Permission is hereby granted, free of charge, to any person obtaining a copy 
of this software and associated documentation files (the "Software"), to deal 
in the Software without restriction, including without limitation the rights 
to use, copy, modify, merge, publish, distribute, sublicense, and/or sell 
copies of the Software, and to permit persons to whom the Software is 
furnished to do so, subject to the following conditions:

The above copyright notice and this permission notice shall be included in 
all copies or substantial portions of the Software.

THE SOFTWARE IS PROVIDED "AS IS", WITHOUT WARRANTY OF ANY KIND, EXPRESS OR 
IMPLIED, INCLUDING BUT NOT LIMITED TO THE WARRANTIES OF MERCHANTABILITY, 
FITNESS FOR A PARTICULAR PURPOSE AND NONINFRINGEMENT. IN NO EVENT SHALL THE 
AUTHORS OR COPYRIGHT HOLDERS BE LIABLE FOR ANY CLAIM, DAMAGES OR OTHER 
LIABILITY, WHETHER IN AN ACTION OF CONTRACT, TORT OR OTHERWISE, ARISING FROM, 
OUT OF OR IN CONNECTION WITH THE SOFTWARE OR THE USE OR OTHER DEALINGS 
IN THE SOFTWARE.
*)
fin := FALSE;
                    
END_ACTION

ACTION TO_DEFAULT_POS_2_active:
                      (*
Copyright (c) 2019 Manuel Goester, Michael Witt, Klaus Kammerer
Institute of Databases and Information Systems, Ulm University, Germany

Permission is hereby granted, free of charge, to any person obtaining a copy 
of this software and associated documentation files (the "Software"), to deal 
in the Software without restriction, including without limitation the rights 
to use, copy, modify, merge, publish, distribute, sublicense, and/or sell 
copies of the Software, and to permit persons to whom the Software is 
furnished to do so, subject to the following conditions:

The above copyright notice and this permission notice shall be included in 
all copies or substantial portions of the Software.

THE SOFTWARE IS PROVIDED "AS IS", WITHOUT WARRANTY OF ANY KIND, EXPRESS OR 
IMPLIED, INCLUDING BUT NOT LIMITED TO THE WARRANTIES OF MERCHANTABILITY, 
FITNESS FOR A PARTICULAR PURPOSE AND NONINFRINGEMENT. IN NO EVENT SHALL THE 
AUTHORS OR COPYRIGHT HOLDERS BE LIABLE FOR ANY CLAIM, DAMAGES OR OTHER 
LIABILITY, WHETHER IN AN ACTION OF CONTRACT, TORT OR OTHERWISE, ARISING FROM, 
OUT OF OR IN CONNECTION WITH THE SOFTWARE OR THE USE OR OTHER DEALINGS 
IN THE SOFTWARE.
*)
// get HR to its default position
// needed, if a job multi / single mode batch job will be executed after ths batch
IF HR.sCBack = FALSE THEN
	HR.mCBackward := TRUE;
ELSE 
	HR.mCBackward := FALSE;
	// set tower vertical position to max UP as well as horizontal position max RIGHT
	IF HR.sHorizontal = FALSE THEN
		HR.mHorizontalRight := TRUE;
	ELSE
		HR.mHorizontalRight := FALSE;
		HR.cX := 0;
	END_IF
	
	IF HR.sVertical = FALSE THEN
		HR.mVerticalUp := TRUE;
	ELSE
		HR.mVerticalUp := FALSE;
		HR.cY := 0;
	END_IF
END_IF

IF HR.sHorizontal AND HR.sVertical AND HR.sCBack THEN
	// finished
	fin := TRUE;
END_IF
                    
END_ACTION
END_PROGRAM

(* Picks up a workpiece Copyright (c) 2019 Manuel Goester, Michael Witt, Klaus Kammerer Institute of Databases and Information Systems, Ulm University, Germany Permission is hereby granted, free of charge, to any person obtaining a copy of this software and associated documentation files (the "Software"), to deal in the Software without restriction, including without limitation the rights to use, copy, modify, merge, publish, distribute, sublicense, and/or sell copies of the Software, and to permit persons to whom the Software is furnished to do so, subject to the following conditions: The above copyright notice and this permission notice shall be included in all copies or substantial portions of the Software. THE SOFTWARE IS PROVIDED "AS IS", WITHOUT WARRANTY OF ANY KIND, EXPRESS OR IMPLIED, INCLUDING BUT NOT LIMITED TO THE WARRANTIES OF MERCHANTABILITY, FITNESS FOR A PARTICULAR PURPOSE AND NONINFRINGEMENT. IN NO EVENT SHALL THE AUTHORS OR COPYRIGHT HOLDERS BE LIABLE FOR ANY CLAIM, DAMAGES OR OTHER LIABILITY, WHETHER IN AN ACTION OF CONTRACT, TORT OR OTHERWISE, ARISING FROM, OUT OF OR IN CONNECTION WITH THE SOFTWARE OR THE USE OR OTHER DEALINGS IN THE SOFTWARE. *)
FUNCTION_BLOCK HR_TAKE_W
  VAR_INPUT
    w : Workpiece;  (* The workpiece *)
  END_VAR
  VAR
    step : INT := 1;
    hr_move : HR_MOVE;
    fin : BOOL := FALSE;
    stepFin : BOOL := FALSE;
  END_VAR

                  fin := FALSE;
CASE step OF
	1:	// forward
		IF NOT(HR.sCFront) THEN
			HR.mCForward := TRUE;
		ELSE
			HR.mCForward := FALSE;
			step := step + 1;
		END_IF
	2:	// up
		hr_move(x := 0, y := -16);
		stepFin := hr_move.fin;
		IF stepFin THEN
			step := step + 1;
			stepFin := FALSE;
		END_IF
	3:	// step 3: back
		IF NOT(HR.sCBack) THEN
			HR.mCBackward := TRUE;
		ELSE
			HR.mCBackward := FALSE;
			step := step + 1;
		END_IF
	4:	// finished
		fin := TRUE;
		step := 1;
		stepFin := FALSE;	
END_CASE
                
END_FUNCTION_BLOCK

(* Moves VG to certain position Copyright (c) 2019 Manuel Goester, Michael Witt, Klaus Kammerer Institute of Databases and Information Systems, Ulm University, Germany Permission is hereby granted, free of charge, to any person obtaining a copy of this software and associated documentation files (the "Software"), to deal in the Software without restriction, including without limitation the rights to use, copy, modify, merge, publish, distribute, sublicense, and/or sell copies of the Software, and to permit persons to whom the Software is furnished to do so, subject to the following conditions: The above copyright notice and this permission notice shall be included in all copies or substantial portions of the Software. THE SOFTWARE IS PROVIDED "AS IS", WITHOUT WARRANTY OF ANY KIND, EXPRESS OR IMPLIED, INCLUDING BUT NOT LIMITED TO THE WARRANTIES OF MERCHANTABILITY, FITNESS FOR A PARTICULAR PURPOSE AND NONINFRINGEMENT. IN NO EVENT SHALL THE AUTHORS OR COPYRIGHT HOLDERS BE LIABLE FOR ANY CLAIM, DAMAGES OR OTHER LIABILITY, WHETHER IN AN ACTION OF CONTRACT, TORT OR OTHERWISE, ARISING FROM, OUT OF OR IN CONNECTION WITH THE SOFTWARE OR THE USE OR OTHER DEALINGS IN THE SOFTWARE. *)
FUNCTION_BLOCK VG_MOVE_TO_POS
  VAR_INPUT
    x : INT;
    y : INT;
    z : INT;
  END_VAR
  VAR
    xFin : BOOL := FALSE;  (* finish flags *)
    yFin : BOOL := FALSE;
    zFin : BOOL := FALSE;
    fin : BOOL := FALSE;
    xAlreadyCounted : BOOL := FALSE;  (* true, if an impulse coming from the motor has been already counted *)
    yAlreadyCounted : BOOL := FALSE;
    zAlreadyCounted : BOOL := FALSE;
  END_VAR

                  fin := FALSE;
// to handle negative counter values
IF VG.cX < 0 THEN
	VG.cX := 0;
END_IF
IF VG.cY < 0 THEN
	VG.cY := 0;
END_IF
IF VG.cZ < 0 THEN
	VG.cZ := 0;
END_IF

// X AXIS (Forward/Backward)
IF VG.cX = x THEN
	// if counter reached demanded position, we're done
	VG.mHorizontalForward := FALSE;
	VG.mHorizontalBackward := FALSE;
	xFin := TRUE;
ELSE
	xFin := FALSE;
	IF VG.cX < x AND NOT(xFin) THEN
		VG.mHorizontalForward := TRUE;
		VG.mHorizontalBackward := FALSE;
		IF VG.encHorizontal AND NOT(xAlreadyCounted) THEN
			VG.cX := VG.cX + 1;
			xAlreadyCounted := TRUE;
		ELSIF NOT(VG.encHorizontal) THEN
			xAlreadyCounted := FALSE;
		END_IF
	ELSIF VG.cX > x AND NOT(xFin) THEN
		VG.mHorizontalForward := FALSE;
		VG.mHorizontalBackward := TRUE;
		IF VG.encHorizontal AND NOT(xAlreadyCounted) THEN
			VG.cX := VG.cX - 1;
			xAlreadyCounted := TRUE;
		ELSIF NOT(VG.encHorizontal) THEN
			xAlreadyCounted := FALSE;
		END_IF
	END_IF
END_IF

// Y AXIS (Up/Down)
IF VG.cY = y THEN
	// if counter reached demanded position, we're done
	VG.mVerticalUp := FALSE;
	VG.mVerticalDown := FALSE;
	yFin := TRUE;
ELSE
	yFin := FALSE;
	IF VG.cY < y AND NOT(yFin) THEN
		VG.mVerticalDown := TRUE;
		VG.mVerticalUp := FALSE;
		IF VG.encVertical AND NOT(yAlreadyCounted) THEN
			VG.cY := VG.cY + 1;
			yAlreadyCounted := TRUE;
		ELSIF NOT(VG.encVertical) THEN
			yAlreadyCounted := FALSE;
		END_IF
	ELSIF VG.cY > y AND NOT(yFin) THEN
		VG.mVerticalUp := TRUE;
		VG.mVerticalDown := FALSE;
		IF VG.encVertical AND NOT(yAlreadyCounted) THEN
			VG.cY := VG.cY - 1;
			yAlreadyCounted := TRUE;
		ELSIF NOT(VG.encVertical) THEN
			yAlreadyCounted := FALSE;
		END_IF
	END_IF
END_IF

// Z AXIS (Rotation)
IF VG.cZ = z THEN
	// if counter reached demanded position, we're done
	VG.mRotationCClockwise := FALSE;
	VG.mRotationClockwise := FALSE;
	zFin := TRUE;
ELSE
	zFin := FALSE;
	IF VG.cZ < z AND NOT(zFin) THEN
		VG.mRotationCClockwise := TRUE;
		VG.mRotationClockwise := FALSE;
		IF VG.encRotation AND NOT(zAlreadyCounted) THEN
			VG.cZ := VG.cZ + 1;
			zAlreadyCounted := TRUE;
		ELSIF NOT(VG.encRotation) THEN
			zAlreadyCounted := FALSE;
		END_IF
	ELSIF VG.cZ > z AND NOT(zFin) THEN
		VG.mRotationCClockwise := FALSE;
		VG.mRotationClockwise := TRUE;
		IF VG.encRotation AND NOT(zAlreadyCounted) THEN
			VG.cZ := VG.cZ - 1;
			zAlreadyCounted := TRUE;
		ELSIF NOT(VG.encRotation) THEN
			zAlreadyCounted := FALSE;
		END_IF
	END_IF
END_IF

// if x and y axis are finsihed, we're done
IF xFin AND yFin AND zFin THEN
	fin := TRUE;
	RETURN;
END_IF
                
END_FUNCTION_BLOCK

(* HR puts down a workpiece at conveyor Copyright (c) 2019 Manuel Goester, Michael Witt, Klaus Kammerer Institute of Databases and Information Systems, Ulm University, Germany Permission is hereby granted, free of charge, to any person obtaining a copy of this software and associated documentation files (the "Software"), to deal in the Software without restriction, including without limitation the rights to use, copy, modify, merge, publish, distribute, sublicense, and/or sell copies of the Software, and to permit persons to whom the Software is furnished to do so, subject to the following conditions: The above copyright notice and this permission notice shall be included in all copies or substantial portions of the Software. THE SOFTWARE IS PROVIDED "AS IS", WITHOUT WARRANTY OF ANY KIND, EXPRESS OR IMPLIED, INCLUDING BUT NOT LIMITED TO THE WARRANTIES OF MERCHANTABILITY, FITNESS FOR A PARTICULAR PURPOSE AND NONINFRINGEMENT. IN NO EVENT SHALL THE AUTHORS OR COPYRIGHT HOLDERS BE LIABLE FOR ANY CLAIM, DAMAGES OR OTHER LIABILITY, WHETHER IN AN ACTION OF CONTRACT, TORT OR OTHERWISE, ARISING FROM, OUT OF OR IN CONNECTION WITH THE SOFTWARE OR THE USE OR OTHER DEALINGS IN THE SOFTWARE. *)
FUNCTION_BLOCK HR_PUT_W_ON_CONVEYOR
  VAR_INPUT
    w : Workpiece;  (* The workpiece *)
  END_VAR
  VAR
    step : INT := 1;
    hr_move : HR_MOVE;
    fin : BOOL := FALSE;
    stepFin : BOOL := FALSE;
  END_VAR

                  CASE step OF
	1:	// forward
		fin := FALSE;	
		IF NOT(HR.sCFront) THEN
			HR.mCForward := TRUE;
		ELSE
			HR.mCForward := FALSE;
			step := step + 1;
		END_IF
	2:	// down
		hr_move(x := 0 , y := 26);
		stepFin := hr_move.fin; 
		IF stepFin THEN
			step := step + 1;
			stepFin := FALSE;
		END_IF
	3:	// finished
		fin := TRUE;
		step := 1;
END_CASE
	
                
END_FUNCTION_BLOCK

(* Picks up a workpiece from conveyor Copyright (c) 2019 Manuel Goester, Michael Witt, Klaus Kammerer Institute of Databases and Information Systems, Ulm University, Germany Permission is hereby granted, free of charge, to any person obtaining a copy of this software and associated documentation files (the "Software"), to deal in the Software without restriction, including without limitation the rights to use, copy, modify, merge, publish, distribute, sublicense, and/or sell copies of the Software, and to permit persons to whom the Software is furnished to do so, subject to the following conditions: The above copyright notice and this permission notice shall be included in all copies or substantial portions of the Software. THE SOFTWARE IS PROVIDED "AS IS", WITHOUT WARRANTY OF ANY KIND, EXPRESS OR IMPLIED, INCLUDING BUT NOT LIMITED TO THE WARRANTIES OF MERCHANTABILITY, FITNESS FOR A PARTICULAR PURPOSE AND NONINFRINGEMENT. IN NO EVENT SHALL THE AUTHORS OR COPYRIGHT HOLDERS BE LIABLE FOR ANY CLAIM, DAMAGES OR OTHER LIABILITY, WHETHER IN AN ACTION OF CONTRACT, TORT OR OTHERWISE, ARISING FROM, OUT OF OR IN CONNECTION WITH THE SOFTWARE OR THE USE OR OTHER DEALINGS IN THE SOFTWARE. *)
FUNCTION_BLOCK HR_TAKE_W_FROM_CONVEYOR
  VAR_INPUT
    w : Workpiece;
  END_VAR
  VAR
    step : INT := 1;
    hr_move : HR_MOVE;
    fin : BOOL := FALSE;
    stepFin : BOOL := FALSE;
  END_VAR

                  fin := FALSE;
CASE step OF
	1:	// forward if not already there
		IF NOT(HR.sCFront) THEN
			HR.mCForward := TRUE;
		ELSE
			HR.mCForward := FALSE;
			step := step + 1;
		END_IF
	2:	// backwards
		IF HR.lbIn THEN
			HR.mCbBackward := TRUE;
		ELSE
			HR.mCbBackward := FALSE;
			step := step + 1; 
		END_IF
	3:	// up
		hr_move(x := 0, y := -26);
		stepFin := hr_move.fin;
		IF stepFin THEN
			step := step + 1;
			stepFin := FALSE;
		END_IF
	4:	// back
		IF NOT(HR.sCBack) THEN
			HR.mCBackward := TRUE;
		ELSE
			HR.mCBackward := FALSE;
			step := step + 1;
		END_IF
	5:	// finished
		fin := TRUE;
		step := 1;
		stepFin := FALSE;
END_CASE
                
END_FUNCTION_BLOCK

(* Function Block for buring a workpiece in furnace w : Workpiece to be burned Copyright (c) 2019 Manuel Goester, Michael Witt, Klaus Kammerer Institute of Databases and Information Systems, Ulm University, Germany Permission is hereby granted, free of charge, to any person obtaining a copy of this software and associated documentation files (the "Software"), to deal in the Software without restriction, including without limitation the rights to use, copy, modify, merge, publish, distribute, sublicense, and/or sell copies of the Software, and to permit persons to whom the Software is furnished to do so, subject to the following conditions: The above copyright notice and this permission notice shall be included in all copies or substantial portions of the Software. THE SOFTWARE IS PROVIDED "AS IS", WITHOUT WARRANTY OF ANY KIND, EXPRESS OR IMPLIED, INCLUDING BUT NOT LIMITED TO THE WARRANTIES OF MERCHANTABILITY, FITNESS FOR A PARTICULAR PURPOSE AND NONINFRINGEMENT. IN NO EVENT SHALL THE AUTHORS OR COPYRIGHT HOLDERS BE LIABLE FOR ANY CLAIM, DAMAGES OR OTHER LIABILITY, WHETHER IN AN ACTION OF CONTRACT, TORT OR OTHERWISE, ARISING FROM, OUT OF OR IN CONNECTION WITH THE SOFTWARE OR THE USE OR OTHER DEALINGS IN THE SOFTWARE. *)
FUNCTION_BLOCK FUR_BURN
  VAR_INPUT
    w : Workpiece;
  END_VAR
  VAR
    step : INT := 1;
    fin : BOOL := FALSE;
    stepFin : BOOL := FALSE;
    timer : TON;
  END_VAR

                  CASE step OF
	1:	// open door and drive workpiece into furnace
		// reset flag
		fin := FALSE;
		FUR.compressor := TRUE;
		FUR.valveFurnanceDoor := TRUE;
		IF FUR.sFurnanceSliderInside = FALSE THEN
			FUR.mFurnanceSliderIn := TRUE;
		ELSE
			FUR.mFurnanceSliderIn := FALSE;
			FUR.state := FUR_State.FUR_WAGON_INSIDE;
			step := step + 1;
		END_IF
	2:	// burn
		IF FUR.state = FUR_State.FUR_WAGON_INSIDE THEN
			//SM.currW.state := StateEnum.AT_FUR_IN_FUR;
			timer(IN:= TRUE, PT := FUR.currWBurner.format.furDuration);
			FUR.valveFurnanceDoor := FALSE;
			IF NOT(timer.Q = FALSE AND timer.IN) THEN
				// reset timer
				timer(IN:= FALSE);
				FUR.compressor := TRUE;
				FUR.valveFurnanceDoor := TRUE;
				FUR.state := FUR_State.FUR_BURNED;
				step := step + 1;
			END_IF
		END_IF
	3:	// drive slider out
		IF FUR.state = FUR_State.FUR_BURNED THEN
			//SM.currW.state := StateEnum.AT_FUR_IN_WAGON;
			IF FUR.sFurnanceSliderOutside = FALSE THEN
				FUR.mFurnanceSliderOut := TRUE;
			ELSE
				FUR.mFurnanceSliderOut := FALSE;
				FUR.state := FUR_State.FUR_WAGON_OUTSIDE;
				FUR.compressor := FALSE;
				FUR.valveFurnanceDoor := FALSE;
				step := step + 1;
			END_IF
		END_IF
	4:	// finished
		fin := TRUE;
		step := 1;
END_CASE

                
END_FUNCTION_BLOCK

(* Implements the functionality of sorting line *)
FUNCTION_BLOCK SL_FB
  VAR
    trigger : INT;
    puls_temp : INT := 0;
    counter_puls : INT;
    white : BOOL;
    red : BOOL;
    blue : BOOL;
    color_value : DINT;
    rack_white : INT := 0;
    rack_red : INT := 0;
    rack_blue : INT := 0;
    timer : TON;
    passed : BOOL;
    fin : BOOL;
  END_VAR

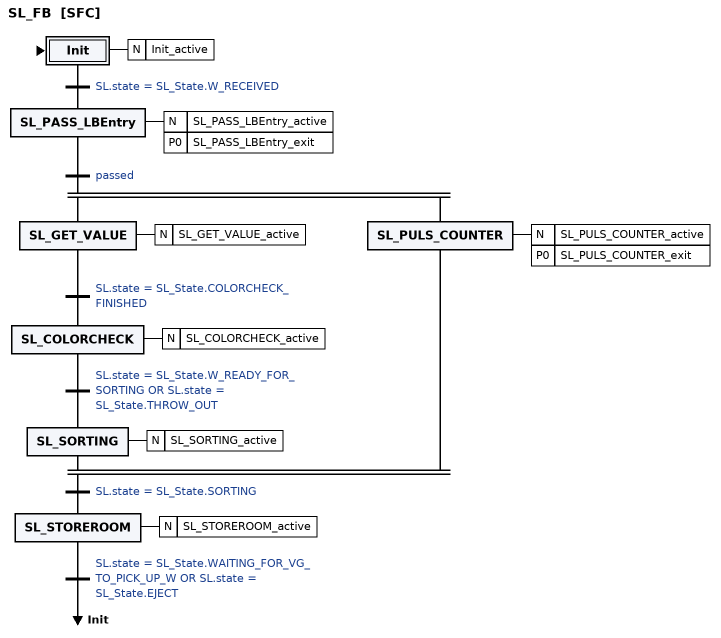
INITIAL_STEP Init:
  Init_active(N);
END_STEP
TRANSITION FROM Init TO SL_PASS_LBEntry
  := SL.state = SL_State.W_RECEIVED;
END_TRANSITION
STEP SL_PASS_LBEntry:
  SL_PASS_LBEntry_active(N);
  SL_PASS_LBEntry_exit(P0);
END_STEP
TRANSITION FROM SL_PASS_LBEntry TO (SL_GET_VALUE, SL_PULS_COUNTER)
  := passed;
END_TRANSITION
STEP SL_GET_VALUE:
  SL_GET_VALUE_active(N);
END_STEP
TRANSITION FROM SL_GET_VALUE TO SL_COLORCHECK
  := SL.state = SL_State.COLORCHECK_FINISHED;
END_TRANSITION
STEP SL_COLORCHECK:
  SL_COLORCHECK_active(N);
END_STEP
TRANSITION FROM SL_COLORCHECK TO SL_SORTING
  := SL.state = SL_State.W_READY_FOR_SORTING OR SL.state = SL_State.THROW_OUT;
END_TRANSITION
STEP SL_SORTING:
  SL_SORTING_active(N);
END_STEP
TRANSITION FROM (SL_SORTING, SL_PULS_COUNTER) TO SL_STOREROOM
  := SL.state = SL_State.SORTING;
END_TRANSITION
STEP SL_PULS_COUNTER:
  SL_PULS_COUNTER_active(N);
  SL_PULS_COUNTER_exit(P0);
END_STEP
STEP SL_STOREROOM:
  SL_STOREROOM_active(N);
END_STEP
TRANSITION FROM SL_STOREROOM TO Init
  := SL.state = SL_State.WAITING_FOR_VG_TO_PICK_UP_W OR SL.state = SL_State.EJECT;
END_TRANSITION

ACTION Init_active:
                      (*
Copyright (c) 2019 Manuel Goester, Michael Witt, Klaus Kammerer
Institute of Databases and Information Systems, Ulm University, Germany

Permission is hereby granted, free of charge, to any person obtaining a copy 
of this software and associated documentation files (the "Software"), to deal 
in the Software without restriction, including without limitation the rights 
to use, copy, modify, merge, publish, distribute, sublicense, and/or sell 
copies of the Software, and to permit persons to whom the Software is 
furnished to do so, subject to the following conditions:

The above copyright notice and this permission notice shall be included in 
all copies or substantial portions of the Software.

THE SOFTWARE IS PROVIDED "AS IS", WITHOUT WARRANTY OF ANY KIND, EXPRESS OR 
IMPLIED, INCLUDING BUT NOT LIMITED TO THE WARRANTIES OF MERCHANTABILITY, 
FITNESS FOR A PARTICULAR PURPOSE AND NONINFRINGEMENT. IN NO EVENT SHALL THE 
AUTHORS OR COPYRIGHT HOLDERS BE LIABLE FOR ANY CLAIM, DAMAGES OR OTHER 
LIABILITY, WHETHER IN AN ACTION OF CONTRACT, TORT OR OTHERWISE, ARISING FROM, 
OUT OF OR IN CONNECTION WITH THE SOFTWARE OR THE USE OR OTHER DEALINGS 
IN THE SOFTWARE.
*)
trigger := 0;
puls_temp := 0;
counter_puls := 0;
white := FALSE;
red := FALSE;
blue := FALSE;

color_value := 4000000;

timer(IN:=FALSE);
fin := FALSE;

SL.mConveyorBelt := TRUE;
                    
END_ACTION

ACTION SL_COLORCHECK_active:
                      (*
Copyright (c) 2019 Manuel Goester, Michael Witt, Klaus Kammerer
Institute of Databases and Information Systems, Ulm University, Germany

Permission is hereby granted, free of charge, to any person obtaining a copy 
of this software and associated documentation files (the "Software"), to deal 
in the Software without restriction, including without limitation the rights 
to use, copy, modify, merge, publish, distribute, sublicense, and/or sell 
copies of the Software, and to permit persons to whom the Software is 
furnished to do so, subject to the following conditions:

The above copyright notice and this permission notice shall be included in 
all copies or substantial portions of the Software.

THE SOFTWARE IS PROVIDED "AS IS", WITHOUT WARRANTY OF ANY KIND, EXPRESS OR 
IMPLIED, INCLUDING BUT NOT LIMITED TO THE WARRANTIES OF MERCHANTABILITY, 
FITNESS FOR A PARTICULAR PURPOSE AND NONINFRINGEMENT. IN NO EVENT SHALL THE 
AUTHORS OR COPYRIGHT HOLDERS BE LIABLE FOR ANY CLAIM, DAMAGES OR OTHER 
LIABILITY, WHETHER IN AN ACTION OF CONTRACT, TORT OR OTHERWISE, ARISING FROM, 
OUT OF OR IN CONNECTION WITH THE SOFTWARE OR THE USE OR OTHER DEALINGS 
IN THE SOFTWARE.
*)
IF color_value > 2000000 AND color_value < 2558000 THEN//weis: 2630000
	TC.batchJobQueue.batchJobs[SL.bIdx].workpieces[SL.wIdx].color := 'white';
	white := TRUE;
	red := FALSE;
	blue := FALSE;
	SL.state := SL_State.W_READY_FOR_SORTING;
END_IF
IF color_value > 2558001 AND color_value < 3000000 THEN//rot: 2801000
	TC.batchJobQueue.batchJobs[SL.bIdx].workpieces[SL.wIdx].color := 'red';
	white := FALSE;
	red := TRUE;
	blue := FALSE;
	SL.state := SL_State.W_READY_FOR_SORTING;
END_IF
IF color_value > 3400000 AND color_value < 3600000 THEN//blau: 3546000
	TC.batchJobQueue.batchJobs[SL.bIdx].workpieces[SL.wIdx].color := 'blue';
	white := FALSE;
	red := FALSE;
	blue := TRUE;
	SL.state := SL_State.W_READY_FOR_SORTING;
END_IF
IF color_value > 3600000 OR color_value < 2000000 THEN//unknown
	TC.batchJobQueue.batchJobs[SL.bIdx].workpieces[SL.wIdx].color := 'unknown';
	white := FALSE;
	red := FALSE;
	blue := FALSE;
	SL.state := SL_State.THROW_OUT; 
END_IF

SL.mConveyorBelt := TRUE;
                    
END_ACTION

ACTION SL_GET_VALUE_active:
                      (*
Copyright (c) 2019 Manuel Goester, Michael Witt, Klaus Kammerer
Institute of Databases and Information Systems, Ulm University, Germany

Permission is hereby granted, free of charge, to any person obtaining a copy 
of this software and associated documentation files (the "Software"), to deal 
in the Software without restriction, including without limitation the rights 
to use, copy, modify, merge, publish, distribute, sublicense, and/or sell 
copies of the Software, and to permit persons to whom the Software is 
furnished to do so, subject to the following conditions:

The above copyright notice and this permission notice shall be included in 
all copies or substantial portions of the Software.

THE SOFTWARE IS PROVIDED "AS IS", WITHOUT WARRANTY OF ANY KIND, EXPRESS OR 
IMPLIED, INCLUDING BUT NOT LIMITED TO THE WARRANTIES OF MERCHANTABILITY, 
FITNESS FOR A PARTICULAR PURPOSE AND NONINFRINGEMENT. IN NO EVENT SHALL THE 
AUTHORS OR COPYRIGHT HOLDERS BE LIABLE FOR ANY CLAIM, DAMAGES OR OTHER 
LIABILITY, WHETHER IN AN ACTION OF CONTRACT, TORT OR OTHERWISE, ARISING FROM, 
OUT OF OR IN CONNECTION WITH THE SOFTWARE OR THE USE OR OTHER DEALINGS 
IN THE SOFTWARE.
*)
IF NOT(SL.lbAfterColorSensor) THEN
	SL.state := SL_State.COLORCHECK_FINISHED;
ELSE
	SL.state := SL_State.W_AT_COLORCHECK;
	IF SL.colorSensor < color_value THEN
		color_value := SL.colorSensor;
	END_IF
END_IF 

SL.mConveyorBelt := TRUE;
                    
END_ACTION

ACTION SL_PASS_LBEntry_active:
                      (*
Copyright (c) 2019 Manuel Goester, Michael Witt, Klaus Kammerer
Institute of Databases and Information Systems, Ulm University, Germany

Permission is hereby granted, free of charge, to any person obtaining a copy 
of this software and associated documentation files (the "Software"), to deal 
in the Software without restriction, including without limitation the rights 
to use, copy, modify, merge, publish, distribute, sublicense, and/or sell 
copies of the Software, and to permit persons to whom the Software is 
furnished to do so, subject to the following conditions:

The above copyright notice and this permission notice shall be included in 
all copies or substantial portions of the Software.

THE SOFTWARE IS PROVIDED "AS IS", WITHOUT WARRANTY OF ANY KIND, EXPRESS OR 
IMPLIED, INCLUDING BUT NOT LIMITED TO THE WARRANTIES OF MERCHANTABILITY, 
FITNESS FOR A PARTICULAR PURPOSE AND NONINFRINGEMENT. IN NO EVENT SHALL THE 
AUTHORS OR COPYRIGHT HOLDERS BE LIABLE FOR ANY CLAIM, DAMAGES OR OTHER 
LIABILITY, WHETHER IN AN ACTION OF CONTRACT, TORT OR OTHERWISE, ARISING FROM, 
OUT OF OR IN CONNECTION WITH THE SOFTWARE OR THE USE OR OTHER DEALINGS 
IN THE SOFTWARE.
*)
IF NOT(SL.lbEntry) AND trigger < 1 THEN
	trigger := trigger + 1;
	SL.state := SL_State.W_AT_LB;
END_IF

IF lbEntry AND trigger >= 1 THEN
	passed := TRUE;
END_IF

SL.mConveyorBelt := TRUE;
                    
END_ACTION

ACTION SL_PASS_LBEntry_exit:
                      (*
Copyright (c) 2019 Manuel Goester, Michael Witt, Klaus Kammerer
Institute of Databases and Information Systems, Ulm University, Germany

Permission is hereby granted, free of charge, to any person obtaining a copy 
of this software and associated documentation files (the "Software"), to deal 
in the Software without restriction, including without limitation the rights 
to use, copy, modify, merge, publish, distribute, sublicense, and/or sell 
copies of the Software, and to permit persons to whom the Software is 
furnished to do so, subject to the following conditions:

The above copyright notice and this permission notice shall be included in 
all copies or substantial portions of the Software.

THE SOFTWARE IS PROVIDED "AS IS", WITHOUT WARRANTY OF ANY KIND, EXPRESS OR 
IMPLIED, INCLUDING BUT NOT LIMITED TO THE WARRANTIES OF MERCHANTABILITY, 
FITNESS FOR A PARTICULAR PURPOSE AND NONINFRINGEMENT. IN NO EVENT SHALL THE 
AUTHORS OR COPYRIGHT HOLDERS BE LIABLE FOR ANY CLAIM, DAMAGES OR OTHER 
LIABILITY, WHETHER IN AN ACTION OF CONTRACT, TORT OR OTHERWISE, ARISING FROM, 
OUT OF OR IN CONNECTION WITH THE SOFTWARE OR THE USE OR OTHER DEALINGS 
IN THE SOFTWARE.
*)
passed := FALSE;
puls_temp := 0;
counter_puls := 0;

                    
END_ACTION

ACTION SL_PULS_COUNTER_active:
                      (*
Copyright (c) 2019 Manuel Goester, Michael Witt, Klaus Kammerer
Institute of Databases and Information Systems, Ulm University, Germany

Permission is hereby granted, free of charge, to any person obtaining a copy 
of this software and associated documentation files (the "Software"), to deal 
in the Software without restriction, including without limitation the rights 
to use, copy, modify, merge, publish, distribute, sublicense, and/or sell 
copies of the Software, and to permit persons to whom the Software is 
furnished to do so, subject to the following conditions:

The above copyright notice and this permission notice shall be included in 
all copies or substantial portions of the Software.

THE SOFTWARE IS PROVIDED "AS IS", WITHOUT WARRANTY OF ANY KIND, EXPRESS OR 
IMPLIED, INCLUDING BUT NOT LIMITED TO THE WARRANTIES OF MERCHANTABILITY, 
FITNESS FOR A PARTICULAR PURPOSE AND NONINFRINGEMENT. IN NO EVENT SHALL THE 
AUTHORS OR COPYRIGHT HOLDERS BE LIABLE FOR ANY CLAIM, DAMAGES OR OTHER 
LIABILITY, WHETHER IN AN ACTION OF CONTRACT, TORT OR OTHERWISE, ARISING FROM, 
OUT OF OR IN CONNECTION WITH THE SOFTWARE OR THE USE OR OTHER DEALINGS 
IN THE SOFTWARE.
*)
//count convoyorbelt buttons
IF SL.mConveyorBelt AND SL.iFeeler THEN //button push
	IF puls_temp = 0 THEN
		counter_puls := counter_puls +1;
	END_IF
	
	puls_temp := puls_temp +1;
END_IF

IF puls_temp > 0 AND SL.mConveyorBelt AND NOT(iFeeler) THEN // button release
	puls_temp := 0;
	counter_puls := counter_puls +1;
END_IF
                    
END_ACTION

ACTION SL_PULS_COUNTER_exit:
                      (*
Copyright (c) 2019 Manuel Goester, Michael Witt, Klaus Kammerer
Institute of Databases and Information Systems, Ulm University, Germany

Permission is hereby granted, free of charge, to any person obtaining a copy 
of this software and associated documentation files (the "Software"), to deal 
in the Software without restriction, including without limitation the rights 
to use, copy, modify, merge, publish, distribute, sublicense, and/or sell 
copies of the Software, and to permit persons to whom the Software is 
furnished to do so, subject to the following conditions:

The above copyright notice and this permission notice shall be included in 
all copies or substantial portions of the Software.

THE SOFTWARE IS PROVIDED "AS IS", WITHOUT WARRANTY OF ANY KIND, EXPRESS OR 
IMPLIED, INCLUDING BUT NOT LIMITED TO THE WARRANTIES OF MERCHANTABILITY, 
FITNESS FOR A PARTICULAR PURPOSE AND NONINFRINGEMENT. IN NO EVENT SHALL THE 
AUTHORS OR COPYRIGHT HOLDERS BE LIABLE FOR ANY CLAIM, DAMAGES OR OTHER 
LIABILITY, WHETHER IN AN ACTION OF CONTRACT, TORT OR OTHERWISE, ARISING FROM, 
OUT OF OR IN CONNECTION WITH THE SOFTWARE OR THE USE OR OTHER DEALINGS 
IN THE SOFTWARE.
*)
counter_puls := 0;
puls_temp := 0;
                    
END_ACTION

ACTION SL_SORTING_active:
                      (*
Copyright (c) 2019 Manuel Goester, Michael Witt, Klaus Kammerer
Institute of Databases and Information Systems, Ulm University, Germany

Permission is hereby granted, free of charge, to any person obtaining a copy 
of this software and associated documentation files (the "Software"), to deal 
in the Software without restriction, including without limitation the rights 
to use, copy, modify, merge, publish, distribute, sublicense, and/or sell 
copies of the Software, and to permit persons to whom the Software is 
furnished to do so, subject to the following conditions:

The above copyright notice and this permission notice shall be included in 
all copies or substantial portions of the Software.

THE SOFTWARE IS PROVIDED "AS IS", WITHOUT WARRANTY OF ANY KIND, EXPRESS OR 
IMPLIED, INCLUDING BUT NOT LIMITED TO THE WARRANTIES OF MERCHANTABILITY, 
FITNESS FOR A PARTICULAR PURPOSE AND NONINFRINGEMENT. IN NO EVENT SHALL THE 
AUTHORS OR COPYRIGHT HOLDERS BE LIABLE FOR ANY CLAIM, DAMAGES OR OTHER 
LIABILITY, WHETHER IN AN ACTION OF CONTRACT, TORT OR OTHERWISE, ARISING FROM, 
OUT OF OR IN CONNECTION WITH THE SOFTWARE OR THE USE OR OTHER DEALINGS 
IN THE SOFTWARE.
*)
SL.mConveyorBelt := TRUE;
IF TC.batchJobQueue.batchJobs[SL.bIdx].workpieces[SL.wIdx].format.colorCheckEnabled THEN
	timer(IN:= TRUE, PT := T#3S);
	IF white AND counter_puls = 35 THEN
		SL.mConveyorBelt := FALSE;
		SL.compressor := TRUE;
		SL.valveFirstEject := TRUE;
	END_IF
	
	IF red AND counter_puls = 45 THEN
		SL.mConveyorBelt := FALSE;
		SL.compressor := TRUE;
		SL.valveSecEject := TRUE;
	END_IF
	
	IF blue AND counter_puls = 55 THEN
		SL.mConveyorBelt := FALSE;
		SL.compressor := TRUE;
		SL.valveThirdEject := TRUE;
	END_IF
	
	IF NOT(timer.Q = FALSE AND timer.IN) THEN
		SL.mConveyorBelt := FALSE;
		SL.compressor := FALSE;	
		SL.valveFirstEject := FALSE;
		SL.valveSecEject := FALSE;
		SL.valveThirdEject := FALSE;
		
		timer(IN:= FALSE);
		
		SL.state := SL_State.SORTING;
	END_IF
ELSE
	timer(IN:= TRUE, PT := T#2S);
	IF counter_puls = 37 THEN
		SL.mConveyorBelt := FALSE;
		SL.compressor := TRUE;
		SL.valveFirstEject := TRUE;
	END_IF
	IF NOT(timer.Q = FALSE AND timer.IN) THEN
		SL.compressor := FALSE;	
		SL.valveFirstEject := FALSE;
		SL.valveSecEject := FALSE;
		SL.valveThirdEject := FALSE;
		
		timer(IN:= FALSE);
		
		SL.state := SL_State.SORTING;
	END_IF
END_IF

                    
END_ACTION

ACTION SL_STOREROOM_active:
                      (*
Copyright (c) 2019 Manuel Goester, Michael Witt, Klaus Kammerer
Institute of Databases and Information Systems, Ulm University, Germany

Permission is hereby granted, free of charge, to any person obtaining a copy 
of this software and associated documentation files (the "Software"), to deal 
in the Software without restriction, including without limitation the rights 
to use, copy, modify, merge, publish, distribute, sublicense, and/or sell 
copies of the Software, and to permit persons to whom the Software is 
furnished to do so, subject to the following conditions:

The above copyright notice and this permission notice shall be included in 
all copies or substantial portions of the Software.

THE SOFTWARE IS PROVIDED "AS IS", WITHOUT WARRANTY OF ANY KIND, EXPRESS OR 
IMPLIED, INCLUDING BUT NOT LIMITED TO THE WARRANTIES OF MERCHANTABILITY, 
FITNESS FOR A PARTICULAR PURPOSE AND NONINFRINGEMENT. IN NO EVENT SHALL THE 
AUTHORS OR COPYRIGHT HOLDERS BE LIABLE FOR ANY CLAIM, DAMAGES OR OTHER 
LIABILITY, WHETHER IN AN ACTION OF CONTRACT, TORT OR OTHERWISE, ARISING FROM, 
OUT OF OR IN CONNECTION WITH THE SOFTWARE OR THE USE OR OTHER DEALINGS 
IN THE SOFTWARE.
*)
IF white AND NOT(SL.lbWhite) THEN
	rack_white := rack_white + 1;
	SL.state := SL_State.WAITING_FOR_VG_TO_PICK_UP_W;
ELSIF red AND NOT(SL.lbRed) THEN
	rack_red := rack_red + 1;
	SL.state := SL_State.WAITING_FOR_VG_TO_PICK_UP_W;
ELSIF blue AND NOT(SL.lbBlue) THEN
	rack_blue := rack_blue + 1;
	SL.state := SL_State.WAITING_FOR_VG_TO_PICK_UP_W;
ELSE
	// no sorting
	SL.state := SL_State.EJECT;
END_IF
// important! --> signals SL_single/multi_MODE PRG that FB is finished
fin := TRUE;
                    
END_ACTION
END_FUNCTION_BLOCK

(* This Function Block gets two workpieces as input and switches their positions in the rack Copyright (c) 2019 Manuel Goester, Michael Witt, Klaus Kammerer Institute of Databases and Information Systems, Ulm University, Germany Permission is hereby granted, free of charge, to any person obtaining a copy of this software and associated documentation files (the "Software"), to deal in the Software without restriction, including without limitation the rights to use, copy, modify, merge, publish, distribute, sublicense, and/or sell copies of the Software, and to permit persons to whom the Software is furnished to do so, subject to the following conditions: The above copyright notice and this permission notice shall be included in all copies or substantial portions of the Software. THE SOFTWARE IS PROVIDED "AS IS", WITHOUT WARRANTY OF ANY KIND, EXPRESS OR IMPLIED, INCLUDING BUT NOT LIMITED TO THE WARRANTIES OF MERCHANTABILITY, FITNESS FOR A PARTICULAR PURPOSE AND NONINFRINGEMENT. IN NO EVENT SHALL THE AUTHORS OR COPYRIGHT HOLDERS BE LIABLE FOR ANY CLAIM, DAMAGES OR OTHER LIABILITY, WHETHER IN AN ACTION OF CONTRACT, TORT OR OTHERWISE, ARISING FROM, OUT OF OR IN CONNECTION WITH THE SOFTWARE OR THE USE OR OTHER DEALINGS IN THE SOFTWARE. *)
FUNCTION_BLOCK HR_SWITCH_WS
  VAR_INPUT
    w1 : Workpiece;  (* first workpiece *)
    w2 : Workpiece;  (* second workpiece *)
  END_VAR
  VAR
    stepFin : BOOL;
    step : INT := 1;
    hr_move_to_pos : HR_MOVE_TO_POS;
    hr_get_w : HR_GET_W;
    hr_take_w : HR_TAKE_W;
    hr_put_w : HR_PUT_W;
    fin : BOOL;
  END_VAR

                  fin := FALSE;
CASE step OF
	1:	// get w1 out of rack and bring it to conveyor
		IF NOT(stepFin) THEN
			hr_get_w(w := w1);
			stepFin := hr_get_w.fin;
		ELSE
			stepFin := FALSE;
			step := step + 1;
		END_IF
	2:	// put down w1 at conveyor
		IF NOT(stepFin) THEN
			hr_put_w();
			stepFin := hr_put_w.fin;
		ELSE
			stepFin := FALSE;
			step := step + 1;
		END_IF
	3:	// move to w2 position in rack
		IF NOT(stepFin) THEN
			hr_move_to_pos(pos := w2.startPos, upOrDown := RackPos.DOWN);	
			stepFin := hr_move_to_pos.fin;
		ELSE
			stepFin := FALSE;
			step := step + 1;
		END_IF
	4:	// pick up w2
		IF NOT(stepFin) THEN
			hr_take_w();
			stepFin := hr_take_w.fin;
		ELSE
			stepFin := FALSE;
			step := step + 1;
		END_IF
	5:	// move to w1 start-position in rack
		IF NOT(stepFin) THEN
			hr_move_to_pos(pos := w1.startPos, upOrDown := RackPos.UP);	
			stepFin := hr_move_to_pos.fin;
		ELSE
			stepFin := FALSE;
			step := step + 1;
		END_IF
	6:	// put down w2 in rack
		IF NOT(stepFin) THEN
			hr_put_w();
			stepFin := hr_put_w.fin;
		ELSE
			stepFin := FALSE;
			step := step + 1;
		END_IF
	7:	// move to conveyor
		IF NOT(stepFin) THEN
			hr_move_to_pos(pos := RackPos.CONVEYOR, upOrDown := RackPos.DOWN);	
			stepFin := hr_move_to_pos.fin;
		ELSE
			stepFin := FALSE;
			step := step + 1;
		END_IF
	8:	// pick up w1 at conveyor
		IF NOT(stepFin) THEN
			hr_take_w();
			stepFin := hr_take_w.fin;
		ELSE
			stepFin := FALSE;
			step := step + 1;
		END_IF
	9:	// move to rack to start-position of w2
		IF NOT(stepFin) THEN
			hr_move_to_pos(pos := w2.startPos, upOrDown := RackPos.UP);	
			stepFin := hr_move_to_pos.fin;
		ELSE
			stepFin := FALSE;
			step := step + 1;
		END_IF
	10:	// put down w1 in rack
		IF NOT(stepFin) THEN
			hr_put_w();
			stepFin := hr_put_w.fin;
		ELSE
			stepFin := FALSE;
			step := step + 1;
		END_IF
	11:	// finished
		fin := TRUE;
		step := 1;
END_CASE
                
END_FUNCTION_BLOCK

CONFIGURATION Application
  RESOURCE Application ON PLC
    VAR_GLOBAL  (* TC *)
      mode_active : ExecutionMode;  (* the mode thats currently active *)
      is_plc_running : BOOL;  (* true if program started *)
      instant_shutdown AT %IX1.7 : BOOL;  (* true if user has selected *)
      batchJobQueue : BatchJobQueue;  (* global batch job queue *)
      currBatchJobIdx : INT := 1;  (* the index in batchJobs of the batch job which is currently running *)
      state : TC_State;  (* state of Task configuration *)
      nullW : Workpiece;  (* This is a workpiece being used as an NULL object in Java *)
      nullB : BatchJob;  (* This is a BatchJob being used as an NULL object in Java *)
    END_VAR
    VAR_GLOBAL  (* SM *)
      currW : Workpiece;  (* SM = single mode current workpiece being processed in single mode *)
    END_VAR
    VAR_GLOBAL  (* HR *)
      sHorizontal AT %IX0.0 : BOOL;  (* ------------------------------------------------------------------------------------// --------------------------------------INPUTS----------------------------------------// ------------------------------------------------------------------------------------// *)
      lbIn AT %IX0.1 : BOOL;
      lbOut AT %IX0.2 : BOOL;
      sVertical AT %IX0.3 : BOOL;
      sCFront AT %IX0.4 : BOOL;
      sCBack AT %IX0.5 : BOOL;
      encHorizontal AT %IX1.1 : BOOL;
      encVertical AT %IX1.2 : BOOL;
      mCbForward AT %QX0.0 : BOOL;  (* ------------------------------------------------------------------------------------// --------------------------------------OUTPUTS---------------------------------------// ------------------------------------------------------------------------------------// *)
      mCbBackward AT %QX0.1 : BOOL;
      mHorizontalLeft AT %QX0.2 : BOOL;
      mHorizontalRight AT %QX0.3 : BOOL;
      mVerticalDown AT %QX0.4 : BOOL;
      mVerticalUp AT %QX0.5 : BOOL;
      mCForward AT %QX0.6 : BOOL;
      mCBackward AT %QX0.7 : BOOL;
      state : HR_State;  (* ------------------------------------------------------------------------------------// ------------------------------------PROGRAM VARS------------------------------------// ------------------------------------------------------------------------------------// the state in which HR currently is *)
      started_btn_is_pressed : BOOL;  (* true if the start button at Visu is pressed *)
      any_motor_running : BOOL;  (* true if any motor of HR is running *)
      decidedToTakeANewW : BOOL;  (* flag needed for decision making in multi mode *)
      cX : INT;  (* these counters define the current position of HR *)
      cY : INT;
      bIdx : INT;  (* current BatchJob and workpiece index being processed at HR *)
      wIdx : INT;
      currW : Workpiece;
    END_VAR
    VAR_GLOBAL  (* FUR *)
      sRaPosSucker AT %IX300.0 : BOOL;  (* ------------------------------------------------------------------------------------// --------------------------------------INPUTS----------------------------------------// ------------------------------------------------------------------------------------// *)
      sRaPosConveyorBelt AT %IX300.1 : BOOL;
      lbConveyorBelt AT %IX300.2 : BOOL;
      sRaPosSaw AT %IX300.3 : BOOL;
      sSuckerPosRa AT %IX300.4 : BOOL;
      sFurnanceSliderInside AT %IX300.5 : BOOL;
      sFurnanceSliderOutside AT %IX300.6 : BOOL;
      sSuckerPosFF AT %IX300.7 : BOOL;
      lbFurnance AT %IX301.0 : BOOL;
      mRaClockwise AT %QX40.0 : BOOL;  (* ------------------------------------------------------------------------------------// --------------------------------------OUTPUTS---------------------------------------// ------------------------------------------------------------------------------------// *)
      mRaCClockwise AT %QX40.1 : BOOL;
      mConveyorBeltForward AT %QX40.2 : BOOL;
      mSaw AT %QX40.3 : BOOL;
      mFurnanceSliderIn AT %QX40.4 : BOOL;
      mFurnanceSliderOut AT %QX40.5 : BOOL;
      mSuckertoFurnance AT %QX40.6 : BOOL;
      mSuckertoRa AT %QX40.7 : BOOL;
      compressor AT %QX41.0 : BOOL;  (* lightFurnance --> NOT ASSIGNED *)
      valveVacuum AT %QX41.1 : BOOL;
      valveLowering AT %QX41.2 : BOOL;
      valveFurnanceDoor AT %QX41.3 : BOOL;
      valveSlider AT %QX41.4 : BOOL;
      any_motor_running : BOOL;  (* ------------------------------------------------------------------------------------// ------------------------------------PROGRAM VARS------------------------------------// ------------------------------------------------------------------------------------// true if any motor/compressor of FUR is running *)
      state : FUR_State;  (* the state in which FUR currently is *)
      bIdxBurner : INT;  (* BatchJob index in BatchJobQueue *)
      bIdxSuccer : INT;
      bIdxSaw : INT;
      wIdxBurner : INT;  (* workpiece index in current BatchJob *)
      wIdxSuccer : INT;
      wIdxSaw : INT;
      currWBurner : Workpiece;  (* current workpieces *)
      currWSuccer : Workpiece;
      currWSaw : Workpiece;
    END_VAR
    VAR_GLOBAL  (* SL *)
      iFeeler AT %IX301.1 : BOOL;  (* ------------------------------------------------------------------------------------// --------------------------------------INPUTS----------------------------------------// ------------------------------------------------------------------------------------// *)
      lbEntry AT %IX301.2 : BOOL;
      lbAfterColorSensor AT %IX301.3 : BOOL;
      colorSensor AT %ID37 : DINT;  (* analog *)
      lbWhite AT %IX301.5 : BOOL;
      lbRed AT %IX301.6 : BOOL;
      lbBlue AT %IX301.7 : BOOL;
      mConveyorBelt AT %QX41.5 : BOOL;  (* ------------------------------------------------------------------------------------// --------------------------------------OUTPUTS---------------------------------------// ------------------------------------------------------------------------------------// *)
      compressor AT %QX41.6 : BOOL;
      valveFirstEject AT %QX41.7 : BOOL;
      valveSecEject AT %QX41.7 : BOOL;
      valveThirdEject AT %QX41.7 : BOOL;
      any_motor_running : BOOL;  (* ------------------------------------------------------------------------------------// ------------------------------------PROGRAM VARS------------------------------------// ------------------------------------------------------------------------------------// true if any motor or compressor of SL is running *)
      state : SL_State;  (* the state in which SL currently is *)
      bIdx : INT;  (* current BatchJob and workpiece index being processed at SL *)
      wIdx : INT;
      currW : Workpiece;
    END_VAR
    VAR_GLOBAL  (* VG *)
      sVertical AT %IX0.6 : BOOL;  (* ------------------------------------------------------------------------------------// --------------------------------------INPUTS----------------------------------------// ------------------------------------------------------------------------------------// s = switch *)
      sHorizontal AT %IX0.7 : BOOL;
      sRotation AT %IX1.0 : BOOL;
      encVertical AT %IX1.3 : BOOL;  (* enc = encoder *)
      encHorizontal AT %IX1.4 : BOOL;
      encRotation AT %IX1.5 : BOOL;
      mVerticalUp AT %QX1.0 : BOOL;  (* ------------------------------------------------------------------------------------// --------------------------------------OUTPUTS---------------------------------------// ------------------------------------------------------------------------------------// m = motor *)
      mVerticalDown AT %QX1.1 : BOOL;
      mHorizontalBackward AT %QX1.2 : BOOL;
      mHorizontalForward AT %QX1.3 : BOOL;
      mRotationClockwise AT %QX1.4 : BOOL;
      mRotationCClockwise AT %QX1.5 : BOOL;
      compressor AT %QX1.6 : BOOL;
      valve AT %QX1.7 : BOOL;
      state : VG_State;  (* ------------------------------------------------------------------------------------// ------------------------------------PROGRAM VARS------------------------------------// ------------------------------------------------------------------------------------// the state in which VG currently is *)
      any_motor_running : BOOL;  (* true if any motor of VG is running *)
      storeW : BOOL;  (* flag used for decision making in multi mode *)
      cX : INT;  (* counters defining the current position of VG *)
      cY : INT;
      cZ : INT;
      bIdx : INT;  (* current BatchJob and workpiece index being processed at VG *)
      wIdx : INT;
      currW : Workpiece;
    END_VAR
    TASK MainTask(INTERVAL := T#4ms, PRIORITY := 0);
    TASK EtherCAT_Master(INTERVAL := T#4ms, PRIORITY := 0);
    TASK VISU_TASK(INTERVAL := T#100ms, PRIORITY := 31);
    PROGRAM EtherCAT_Master.EtherCAT_Task WITH MainTask : EtherCAT_Master.EtherCAT_Task;
    PROGRAM MAIN WITH MainTask : MAIN;
    PROGRAM EtherCAT_Master.EtherCAT_Task WITH EtherCAT_Master : EtherCAT_Master.EtherCAT_Task;
    PROGRAM VisuElems.Visu_Prg WITH VISU_TASK : VisuElems.Visu_Prg;
  END_RESOURCE
END_CONFIGURATION
